SUBAPPLICATION LinksRechts_T_FF (* Subapplication Type *)
  (* Standard: 61499-2 *)
  (* Version 1.0, 2025-05-06, franz *)
  PACKAGE FBs::Uebungen::Uebung_006a3;
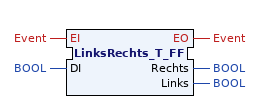
  EVENT_INPUT
    EI;
  END_EVENT
  EVENT_OUTPUT
    EO;
  END_EVENT
  VAR_INPUT
    DI : BOOL;
  END_VAR
  VAR_OUTPUT
    Rechts : BOOL;
    Links : BOOL;
  END_VAR
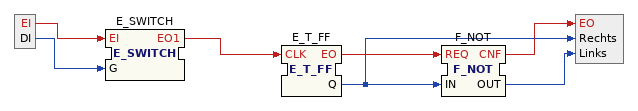
  FBS
    E_T_FF : E_T_FF;
    E_SWITCH : E_SWITCH;
    F_NOT : F_NOT;
  END_FBS
  EVENT_CONNECTIONS
    E_T_FF.EO TO F_NOT.REQ;
    EI TO E_SWITCH.EI;
    F_NOT.CNF TO EO;
    E_SWITCH.EO1 TO E_T_FF.CLK;
  END_CONNECTIONS
  DATA_CONNECTIONS
    E_T_FF.Q TO F_NOT.IN;
    E_T_FF.Q TO Rechts;
    DI TO E_SWITCH.G;
    F_NOT.OUT TO Links;
  END_CONNECTIONS
END_SUBAPPLICATION
